// TIA Portal project "Girello" (V16)

(* hardware
DEVICE "S7-1200 station_1"  S7-1200 Station
   slot 0: "Telaio di montaggio_0"  S7-1200 Rack  Rack  V1.0
   slot 1: "PLC_1"  CPU 1214C DC/DC/DC  6ES7 214-1AG40-0XB0  V4.1
*)

// ===== PLC "PLC_1"  CPU 1214C DC/DC/DC =====

VAR_GLOBAL   // PLC tag table "Tabella delle variabili standard"
   "START_1" AT %I0.0 : Bool;
   "S1_1" AT %I0.1 : Bool;
   "S2_1" AT %I0.2 : Bool;
   "START_2" AT %I0.4 : Bool;
   "S1_2" AT %I0.5 : Bool;
   "S2_2" AT %I0.6 : Bool;
   "M_left_1" AT %Q0.0 : Bool;
   "M_left_2" AT %Q0.1 : Bool;
END_VAR

VAR_GLOBAL CONSTANT   // PLC tag table "Tabella delle variabili standard"
   "TEMPO_TRASCORSO_T1_Girello1" : Time := T#3s;
   "TEMPO_TRASCORSO_T2_Girello2" : Time := T#5s;
END_VAR

DATA_BLOCK "Girello_DB_1"   // DB1
{ S7_Optimized_Access := 'TRUE' }
VERSION : 0.1
// stored: InstanceOfName Girello
"Girello"
BEGIN
END_DATA_BLOCK

DATA_BLOCK "Girello_DB_2"   // DB2
{ S7_Optimized_Access := 'TRUE' }
VERSION : 0.1
// stored: InstanceOfName Girello
"Girello"
BEGIN
END_DATA_BLOCK

FUNCTION_BLOCK "Girello"   // FB1, LAD
{ S7_Optimized_Access := 'TRUE' }
VERSION : 0.1
   VAR_INPUT
      START : Bool;
      S1 : Bool;
      S2 : Bool;
      TEMPO_TRASCORSO : Time;
   END_VAR
   VAR_OUTPUT
      M_left : Bool;
   END_VAR
   VAR RETAIN
      HOME : Bool := true;
      ROTATE_TO_LEFT_1 : Bool;
      POSITION_S2 : Bool;
      ROTATE_TO_LEFT_2 : Bool;
   END_VAR
   VAR
      IEC_Timer_0_Instance : TON_TIME;
   END_VAR
BEGIN

REGION Network 1
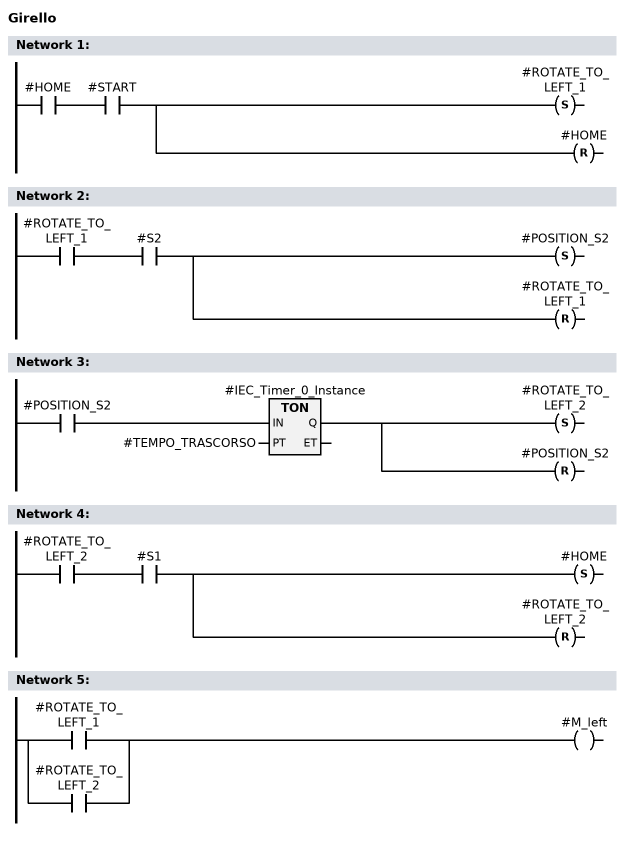
   RUNG wire#powerrail
      Contact( #HOME )
      Contact( #START )
      wire#w1
      S_Coil( #ROTATE_TO_LEFT_1 )
   END_RUNG
   RUNG wire#w1
      R_Coil( #HOME )
   END_RUNG
   // the same network as SCL:
   IF #HOME AND #START THEN
       #ROTATE_TO_LEFT_1 := TRUE;
       #HOME := FALSE;
   END_IF;
END_REGION

REGION Network 2
   RUNG wire#powerrail
      Contact( #ROTATE_TO_LEFT_1 )
      Contact( #S2 )
      wire#w1
      S_Coil( #POSITION_S2 )
   END_RUNG
   RUNG wire#w1
      R_Coil( #ROTATE_TO_LEFT_1 )
   END_RUNG
   // the same network as SCL:
   IF #ROTATE_TO_LEFT_1 AND #S2 THEN
       #POSITION_S2 := TRUE;
       #ROTATE_TO_LEFT_1 := FALSE;
   END_IF;
END_REGION

REGION Network 3
   #IEC_Timer_0_Instance(IN := #POSITION_S2, PT := #TEMPO_TRASCORSO);   // TON
   IF #IEC_Timer_0_Instance.Q THEN
       #ROTATE_TO_LEFT_2 := TRUE;
       #POSITION_S2 := FALSE;
   END_IF;
END_REGION

REGION Network 4
   RUNG wire#powerrail
      Contact( #ROTATE_TO_LEFT_2 )
      Contact( #S1 )
      wire#w1
      S_Coil( #HOME )
   END_RUNG
   RUNG wire#w1
      R_Coil( #ROTATE_TO_LEFT_2 )
   END_RUNG
   // the same network as SCL:
   IF #ROTATE_TO_LEFT_2 AND #S1 THEN
       #HOME := TRUE;
       #ROTATE_TO_LEFT_2 := FALSE;
   END_IF;
END_REGION

REGION Network 5
   RUNG wire#powerrail
      Contact( #ROTATE_TO_LEFT_1 )
      wire#w1
      Coil( #M_left )
   END_RUNG
   RUNG wire#powerrail
      Contact( #ROTATE_TO_LEFT_2 )
   END_RUNG wire#w1
   // the same network as SCL:
   #M_left := #ROTATE_TO_LEFT_1 OR #ROTATE_TO_LEFT_2;
END_REGION
END_FUNCTION_BLOCK

ORGANIZATION_BLOCK "Main"   // OB1, LAD, ProgramCycle
TITLE = "Main Program Sweep (Cycle)"
{ S7_Optimized_Access := 'TRUE' }
VERSION : 0.1
   VAR_INPUT
      Initial_Call : Bool;   // Initial call of this OB
      Remanence : Bool;   // =True, if remanent data are available
   END_VAR
BEGIN
END_ORGANIZATION_BLOCK

ORGANIZATION_BLOCK "Cyclic_Interrupt_50ms"   // OB30, LAD, CyclicInterrupt
{ S7_Optimized_Access := 'TRUE' }
VERSION : 0.1
   VAR_INPUT
      Initial_Call : Bool;   // Initial call of this OB
      Event_Count : Int;   // Events discarded
   END_VAR
BEGIN

REGION Network 1
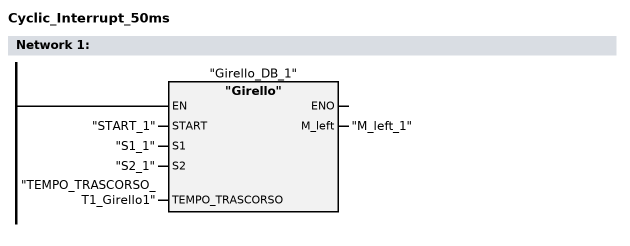
   RUNG wire#powerrail
      "Girello_DB_1"(START := "START_1", S1 := "S1_1", S2 := "S2_1", TEMPO_TRASCORSO := "TEMPO_TRASCORSO_T1_Girello1", M_left => "M_left_1")
   END_RUNG
   // the same network as SCL:
   "Girello_DB_1"(START := "START_1",   // "Girello"
                  S1 := "S1_1",
                  S2 := "S2_1",
                  TEMPO_TRASCORSO := "TEMPO_TRASCORSO_T1_Girello1",
                  M_left => "M_left_1");
END_REGION
END_ORGANIZATION_BLOCK

ORGANIZATION_BLOCK "Cyclic_Interrupt_100ms"   // OB31, LAD, CyclicInterrupt
{ S7_Optimized_Access := 'TRUE' }
VERSION : 0.1
   VAR_INPUT
      Initial_Call : Bool;   // Initial call of this OB
      Event_Count : Int;   // Events discarded
   END_VAR
BEGIN

REGION Network 1
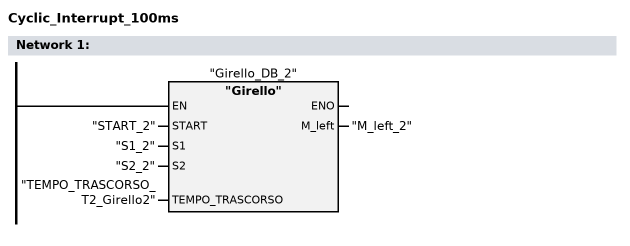
   RUNG wire#powerrail
      "Girello_DB_2"(START := "START_2", S1 := "S1_2", S2 := "S2_2", TEMPO_TRASCORSO := "TEMPO_TRASCORSO_T2_Girello2", M_left => "M_left_2")
   END_RUNG
   // the same network as SCL:
   "Girello_DB_2"(START := "START_2",   // "Girello"
                  S1 := "S1_2",
                  S2 := "S2_2",
                  TEMPO_TRASCORSO := "TEMPO_TRASCORSO_T2_Girello2",
                  M_left => "M_left_2");
END_REGION
END_ORGANIZATION_BLOCK